FUNCTION_BLOCK FB_BSp
VAR_INPUT
	Parameter_init	: ST_BSp_Parameter;
END_VAR
VAR_OUTPUT
	{attribute 'OPC.UA.DA' := '1'}Parameter	: ST_BSp_Parameter;		
	{attribute 'OPC.UA.DA' := '1'}Zustand		: ST_BSp_Zustand;	
	Steuerung	: ST_BSp_Steuerung;
END_VAR
VAR
	Zustandscheck	: FB_BSp_Zustandscheck;

	LeseDaten			: FB_BSp_Input;
(*	IN_Temp_oben		AT %I* : REAL;
	IN_Temp_unten		AT %I* : REAL;
*)	IN_Fuellstandsalarm	AT %I* : BOOL;

	TF_oben		: FB_TF;
	TF_unten	: FB_TF;

END_VAR

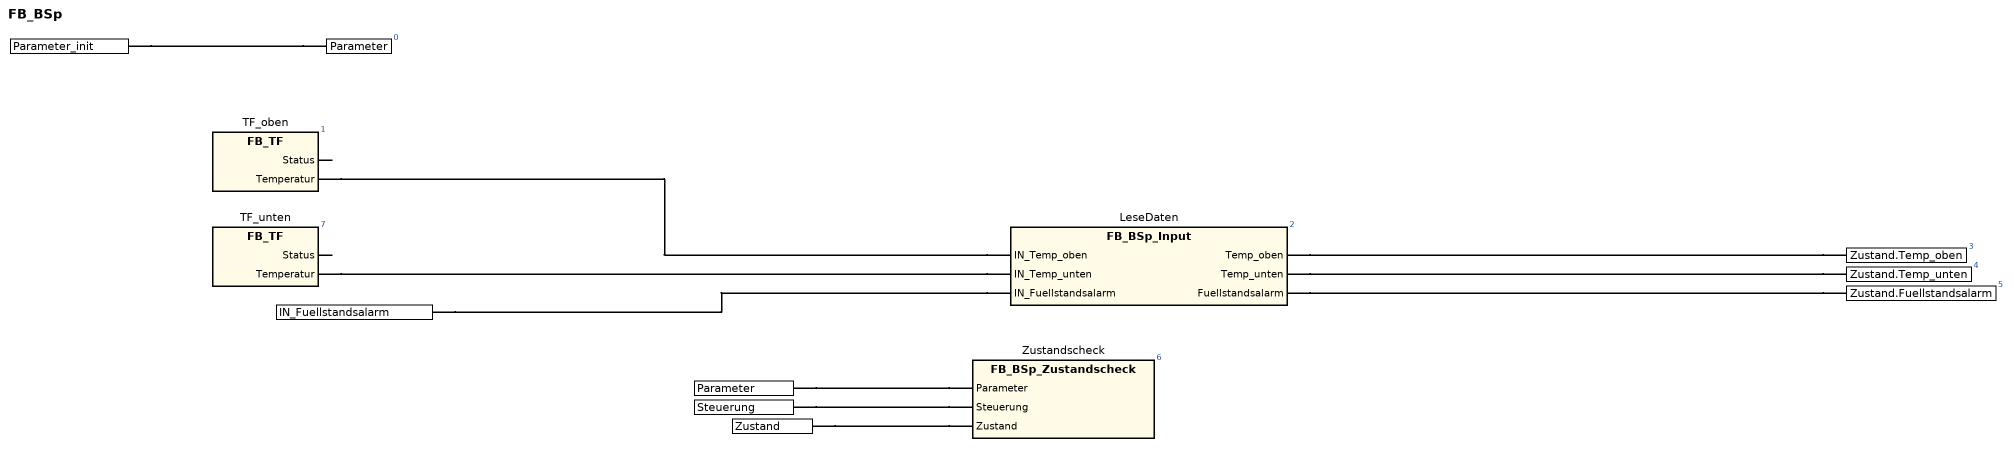
Parameter := Parameter_init;
TF_oben(); // FB_TF
LeseDaten(
    IN_Temp_oben := TF_oben.Temperatur,
    IN_Temp_unten := TF_unten.Temperatur,
    IN_Fuellstandsalarm := IN_Fuellstandsalarm); // FB_BSp_Input
Zustand.Temp_oben := LeseDaten.Temp_oben;
Zustand.Temp_unten := LeseDaten.Temp_unten;
Zustand.Fuellstandsalarm := LeseDaten.Fuellstandsalarm;
Zustandscheck(Parameter := Parameter, Steuerung := Steuerung, Zustand := Zustand); // FB_BSp_Zustandscheck
TF_unten(); // FB_TF

END_FUNCTION_BLOCK

(* stored: Version 1.1.0.1, ProductVersion 3.1.4024.9
   POU FB_BSp: Id {5a89211b-6641-4b16-b689-1ece77736fba}, SpecialFunc None *)
